// SIMATIC S7-200 project (STEP 7-Micro/WIN), CPU 221 REL 01.10

ORGANIZATION_BLOCK 主程序:OB1
TITLE=程序注释
BEGIN
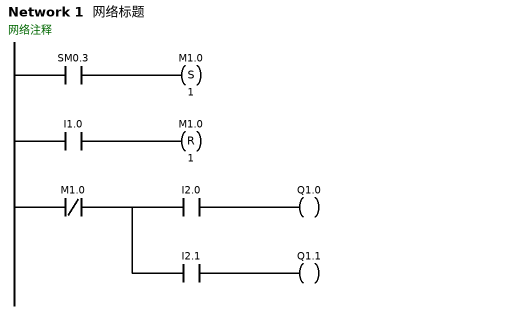
Network 1 // 网络标题
// 网络注释
// (network saved uncompiled; LAD cells follow)
// row 0: c0 -| |- SM0.3  c1 -(S) M1.0, 1
// row 1: c0 -| |- I1.0  c1 -(R) M1.0, 1
// row 2: c0 -|/|- M1.0 v  c1 -| |- I2.0  c2 -( ) Q1.0
// row 3: c0 ^  c1 -| |- I2.1  c2 -( ) Q1.1
END_ORGANIZATION_BLOCK
